FUNCTION_BLOCK ButtonTimer (* Composite Function Block Type *)
  (* Standard: 61499-2 *)
  (* Version 0.0, 5/18/2015, trauscher, nxtControl GmbH, template *)
  PACKAGE Loytec.Automation;
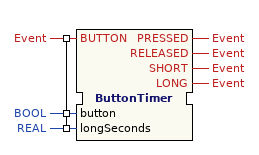
  EVENT_INPUT
    BUTTON WITH button, longSeconds; (* Button event *)
  END_EVENT
  EVENT_OUTPUT
    PRESSED; (* Event when button is pressed *)
    RELEASED; (* Event when button is released *)
    SHORT; (* Event when short press is detected *)
    LONG; (* Event when long press is detected *)
  END_EVENT
  VAR_INPUT
    button : BOOL; (* Button input *)
    longSeconds : REAL; (* Time for long press *)
  END_VAR
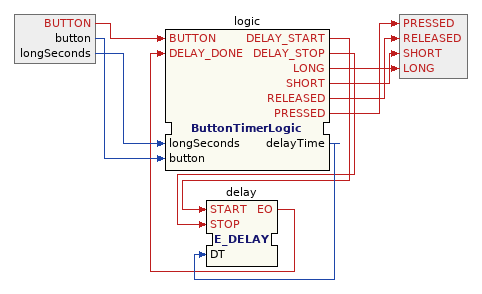
  FBS
    logic : ButtonTimerLogic;
    delay : E_DELAY;
  END_FBS
  EVENT_CONNECTIONS
    BUTTON TO logic.BUTTON;
    logic.DELAY_START TO delay.START;
    logic.DELAY_STOP TO delay.STOP;
    delay.EO TO logic.DELAY_DONE;
    logic.LONG TO LONG;
    logic.SHORT TO SHORT;
    logic.RELEASED TO RELEASED;
    logic.PRESSED TO PRESSED;
  END_CONNECTIONS
  DATA_CONNECTIONS
    logic.delayTime TO delay.DT;
    longSeconds TO logic.longSeconds;
    button TO logic.button;
  END_CONNECTIONS
END_FUNCTION_BLOCK
